FUNCTION_BLOCK Conveyor_SL_1_Adp (* Composite Function Block Type *)
  (* Standard: 61499-2 *)
  (* Version 0.0, 4/23/2020, prana, nxtControl GmbH, template *)
  PACKAGE Main;
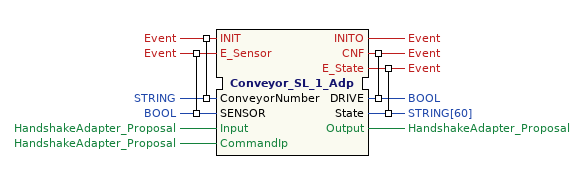
  EVENT_INPUT
    INIT WITH ConveyorNumber; (* Initialization Request *)
    E_Sensor WITH SENSOR;
  END_EVENT
  EVENT_OUTPUT
    INITO; (* Initialization Confirm *)
    CNF WITH DRIVE;
    E_State WITH State;
  END_EVENT
  VAR_INPUT
    ConveyorNumber : STRING;
    SENSOR : BOOL; (* Current value(i) in the named variable array element *)
  END_VAR
  VAR_OUTPUT
    DRIVE : BOOL;
    State : STRING[60];
  END_VAR
  SOCKETS
    Input : HandshakeAdapter_Proposal;
    CommandIp : HandshakeAdapter_Proposal;
  END_SOCKETS
  PLUGS
    Output : HandshakeAdapter_Proposal;
  END_PLUGS
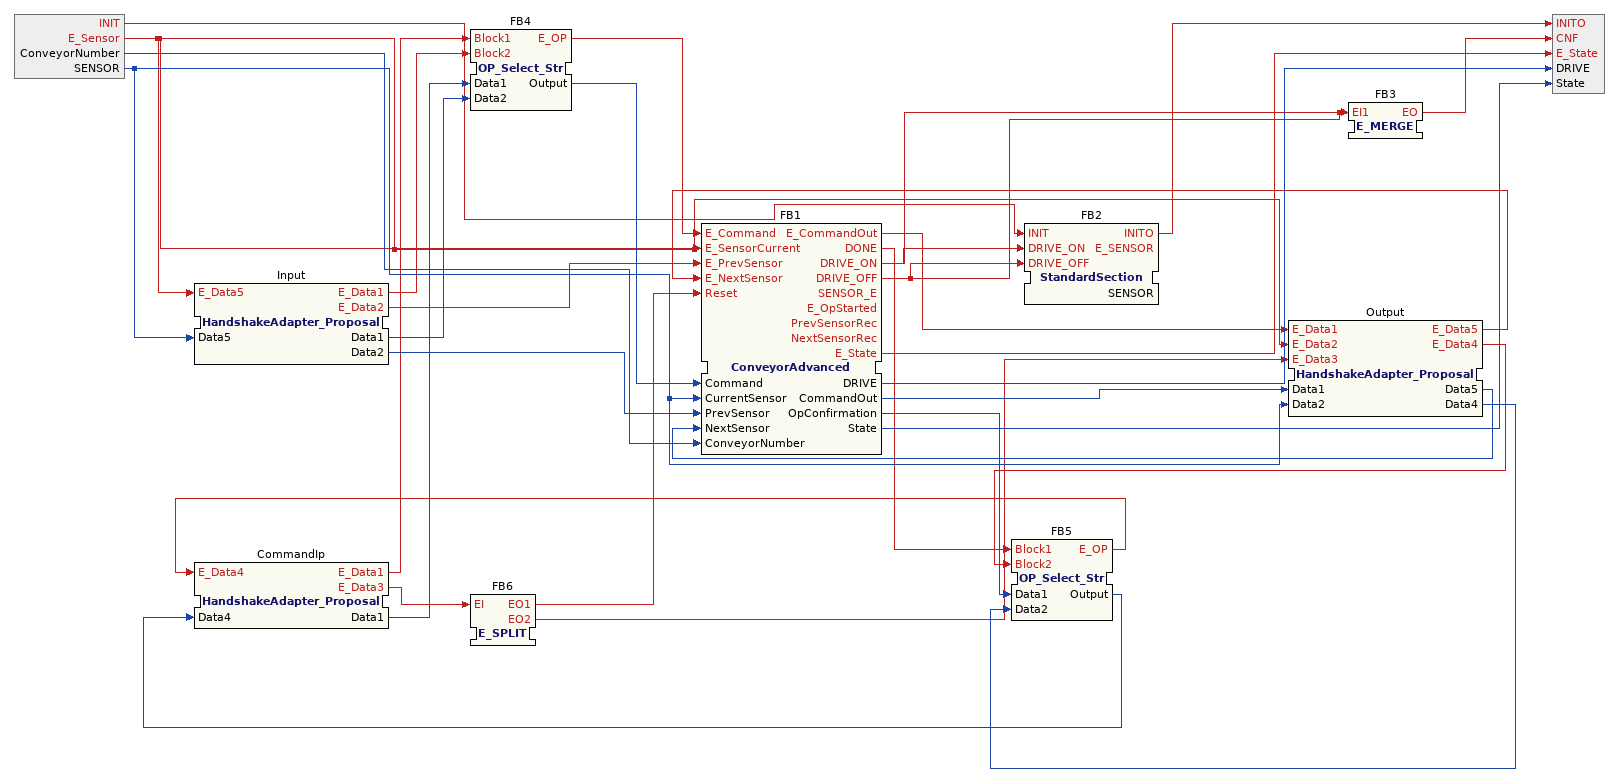
  FBS
    FB2 : StandardSection;
    FB3 : E_MERGE;
    FB1 : ConveyorAdvanced;
    FB4 : OP_Select_Str;
    FB5 : OP_Select_Str;
    FB6 : E_SPLIT;
  END_FBS
  EVENT_CONNECTIONS
    INIT TO FB2.INIT;
    FB1.DRIVE_ON TO FB2.DRIVE_ON;
    FB1.DRIVE_OFF TO FB2.DRIVE_OFF;
    E_Sensor TO FB1.E_SensorCurrent;
    FB3.EO TO CNF;
    FB1.DRIVE_ON TO FB3.EI1;
    FB1.DRIVE_OFF TO FB3.EI1;
    FB4.E_OP TO FB1.E_Command;
    CommandIp.E_Data1 TO FB4.Block1;
    FB1.DONE TO FB5.Block1;
    FB1.E_CommandOut TO Output.E_Data1;
    E_Sensor TO Output.E_Data2;
    Input.E_Data1 TO FB4.Block2;
    Input.E_Data2 TO FB1.E_PrevSensor;
    Output.E_Data5 TO FB1.E_NextSensor;
    Output.E_Data4 TO FB5.Block2;
    FB5.E_OP TO CommandIp.E_Data4;
    E_Sensor TO Input.E_Data5;
    FB2.INITO TO INITO;
    FB1.E_State TO E_State;
    CommandIp.E_Data3 TO FB6.EI;
    FB6.EO1 TO FB1.Reset;
    FB6.EO2 TO Output.E_Data3;
  END_CONNECTIONS
  DATA_CONNECTIONS
    SENSOR TO FB1.CurrentSensor;
    FB1.DRIVE TO DRIVE;
    FB4.Output TO FB1.Command;
    ConveyorNumber TO FB1.ConveyorNumber;
    CommandIp.Data1 TO FB4.Data1;
    FB1.OpConfirmation TO FB5.Data1;
    FB1.CommandOut TO Output.Data1;
    SENSOR TO Output.Data2;
    Input.Data1 TO FB4.Data2;
    Output.Data5 TO FB1.NextSensor;
    Output.Data4 TO FB5.Data2;
    FB5.Output TO CommandIp.Data4;
    SENSOR TO Input.Data5;
    Input.Data2 TO FB1.PrevSensor;
    FB1.State TO State;
  END_CONNECTIONS
END_FUNCTION_BLOCK
